{attribute 'linkalways'} 
{attribute 'no_explicit_call' := 'This FB is a CLASS and must be accessed using methods or properties'}
{attribute 'enable_dynamic_creation'}
FUNCTION_BLOCK FINAL SUB_UINT EXTENDS Node
VAR
	in1 : _UINT(0);
	in2 : _UINT(0);
	out : _UINT(0);
END_VAR

METHOD PUBLIC Clone : I_Node
VAR
	pNode : POINTER TO SUB_UINT;
END_VAR
pNode := __NEW(SUB_UINT);
Clone := pNode^;
END_METHOD

METHOD FB_init : BOOL
VAR_INPUT
	bInitRetains : BOOL; // if TRUE, the retain variables are initialized (warm start / cold start)
	bInCopyCode : BOOL;  // if TRUE, the instance afterwards gets moved into the copy code (online change)
END_VAR
AddInput('in1',THIS^.in1);
AddInput('in2',THIS^.in2);
AddOutput('out', THIS^.out);
END_METHOD

METHOD PROTECTED OnExecute
VAR
END_VAR
out.Value := in1.Value - in2.Value;
END_METHOD

END_FUNCTION_BLOCK

(* stored: Version 1.1.0.1, ProductVersion 3.1.4024.15
   POU SUB_UINT: Id {2bc65def-4dbd-4f9e-bbee-03dbf168522d}, SpecialFunc None
   Folder Constructor: Id {54069e23-174b-4eac-b338-18b1e91f81ab}
   Method Clone: Id {9a40e88c-03cd-4359-8d92-b2a5724f70ec}
   Method FB_init: Id {b1e80d7d-8b3e-43c6-ab13-316c69f20de0}
   Method OnExecute: Id {849e3aa2-f9f0-4187-8569-02761b4b605a} *)
